% RSLogix 500 project PRACTISE-16.RSS, saved by version 8.30.00.16 %
PROJECT "UNTITLED"    % processor: MicroLogix 1000 %

PROGRAM FILES
  LAD 2 "MAIN_PROG"  7 rungs
  LAD 3 "USER_FAULT"  1 rungs
  LAD 4 "HSC_INT"  1 rungs
  LAD 5 "STI_INT"  1 rungs
  LAD 6, 7, 8, 9, 10, 11, 12, 13, 14, 15, 16: only END

DATA FILES
  O0 OUTPUT  1 elements
  I1 INPUT  2 elements
  S2 STATUS  33 elements
  B3 BINARY  32 elements
  T4 TIMER  40 elements
  C5 COUNTER  32 elements
  R6 CONTROL  16 elements
  N7 INTEGER  105 elements

LADDER 2 "MAIN_PROG"
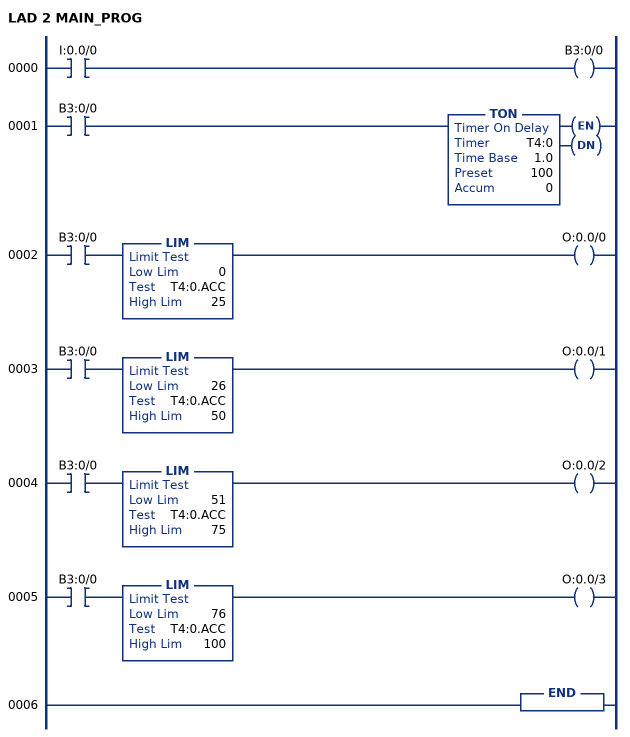
% Rung: 0 %
SOR XIC I:0.0/0 OTE B3:0/0 EOR
% Rung: 1 %
SOR XIC B3:0/0 TON T4:0 1.0 100 0 EOR
% Rung: 2 %
SOR XIC B3:0/0 LIM 0 T4:0.ACC 25 OTE O:0.0/0 EOR
% Rung: 3 %
SOR XIC B3:0/0 LIM 26 T4:0.ACC 50 OTE O:0.0/1 EOR
% Rung: 4 %
SOR XIC B3:0/0 LIM 51 T4:0.ACC 75 OTE O:0.0/2 EOR
% Rung: 5 %
SOR XIC B3:0/0 LIM 76 T4:0.ACC 100 OTE O:0.0/3 EOR
% Rung: 6 %
SOR END EOR

DATA TABLE (non-zero values as saved)
DATA T4
% .PRE .ACC %
% T4:0 % 100 0
